{attribute 'no_check'}
FUNCTION_BLOCK Ax_BrakeCopperIO 
VAR_OUTPUT CONSTANT
END_VAR
VAR_INPUT
END_VAR
VAR_OUTPUT	
	Overtemperature									AT  %I* : BOOL;
	I2T_Error										AT  %I* : BOOL;
	I2T_Warning										AT  %I* : BOOL;
	Overvoltage										AT  %I* : BOOL;
	Undervoltage									AT  %I* : BOOL;
	CopperOn										AT  %I* : BOOL;
	DCLinkVoltage									AT  %I* : UDINT;
	ResistorCurrent									AT  %I* : DINT;
	DutCycle										AT  %I* : USINT;
END_VAR
VAR
{attribute 'hide'}
END_VAR

(* Ax_BrakeCopperIO						*)
(****************************************)
	
(* Work objects ****************************************)
	;
(*******************************************************)

END_FUNCTION_BLOCK

(* stored: Version 1.1.0.1, ProductVersion 3.1.4024.12
   POU Ax_BrakeCopperIO: Id {91b3d4b5-76e1-4aef-be35-d3492cdf7ca4}, SpecialFunc None *)
